FUNCTION_BLOCK FB_FallibleLREAL IMPLEMENTS I_FallibleLREAL
VAR
    bError : BOOL;
    sErrorMsg : T_MaxString;
    fVal : LREAL;
END_VAR

METHOD ClearError

bError := FALSE;
sErrorMsg := '';
END_METHOD

METHOD GetError : BOOL

GetError := bError;
END_METHOD

METHOD GetErrorMsg : Tc2_System.T_MaxString

GetErrorMsg := sErrorMsg;
END_METHOD


METHOD SetError
VAR_INPUT
    sMsg	: Tc2_System.T_MaxString;
END_VAR

bError := TRUE;
sErrorMsg := sMsg;
END_METHOD

PROPERTY Val : LREAL
GET

Val := fVal;
END_GET
SET

fVal := Val;
END_SET
END_PROPERTY

END_FUNCTION_BLOCK

(* stored: Version 1.1.0.1, ProductVersion 3.1.4022.18
   POU FB_FallibleLREAL: Id {5abdc9d0-8a51-408d-9fe6-86a083d1b2a5}, SpecialFunc None
   Method ClearError: Id {58eb6dba-a846-4edd-9264-140e35721fb7}
   Method GetError: Id {e19b6b59-0f9f-4ee9-a5e6-0b73e7628c90}
   Method GetErrorMsg: Id {de67690c-70e9-488d-8a80-288b15210c42}
   Method SetError: Id {3dc8d9a6-9226-4cd8-80ee-ac051b77d47d}
   Property Val: Id {fc1f1cbd-cf1e-4f31-a752-9206efe27500}
   Get Get: Id {3464c393-590e-4402-92b1-141fce4ea36a}
   Set Set: Id {ed169f05-bb80-4af5-b408-f0efc1b7eee3} *)
